FUNCTION_BLOCK FB_DataCollectionSequence
VAR
    iSystemCalibration : I_SystemCalibration;
    iResetSequence : I_ResetSequence;
    iTriggerManager : I_TriggerManager;

    eSequence : E_DataCollectionSequenceStep;
END_VAR


// Run our sequence here

CASE eSequence OF
    E_DataCollectionSequenceStep.WaitingForStart :
        // Do nothing

    E_DataCollectionSequenceStep.WaitingForInitialTrigger :

    E_DataCollectionSequenceStep.CalculateTimeToNextPoint :

    E_DataCollectionSequenceStep.AccelerateToScanningSpeed :

    E_DataCollectionSequenceStep.OperateAtScanningSpeedMakingMinuteAdjustments :

    E_DataCollectionSequenceStep.GoToNextRow :

    E_DataCollectionSequenceStep.WaitingForTriggerToStartNewRow :

    E_DataCollectionSequenceStep.Error :
        // Do nothing
    E_DataCollectionSequenceStep.Done :
        // Do nothing
END_CASE

//FB_Init is always available implicitly and it is used primarily for initialization.
//The return value is not evaluated. For a specific influence, you can also declare the
//methods explicitly and provide additional code there with the standard initialization
//code. You can evaluate the return value.
METHOD FB_Init: BOOL
VAR_INPUT
    bInitRetains: BOOL; // TRUE: the retain variables are initialized (reset warm / reset cold)
    bInCopyCode: BOOL;  // TRUE: the instance will be copied to the copy code afterward (online change)
    iSystemCalibration : I_SystemCalibration;
    iResetSequence : I_ResetSequence;
    iTriggerManager : I_TriggerManager;
END_VAR
THIS^.iSystemCalibration := iSystemCalibration;
THIS^.iResetSequence := iResetSequence;
THIS^.iTriggerManager := iTriggerManager;
END_METHOD

METHOD PRIVATE GetDataCollectionSequenceStep : E_DataCollectionSequenceStep
GetDataCollectionSequenceStep := THIS^.eSequence;
END_METHOD

METHOD PUBLIC IsRunningSequence : BOOL
IsRunningSequence := (GetDataCollectionSequenceStep() <> E_DataCollectionSequenceStep.WaitingForStart) AND
                     (GetDataCollectionSequenceStep() <> E_DataCollectionSequenceStep.Error) AND
                     (GetDataCollectionSequenceStep() <> E_DataCollectionSequenceStep.Done);
END_METHOD


METHOD PUBLIC Start
VAR_OUTPUT
    bError : BOOL;
    sErrorString : T_MaxString;
END_VAR

IF NOT iSystemCalibration.IsCalibrated() THEN
    bError := TRUE;
    sErrorString := 'Can$'t start data collection sequence. System is not calibrated';
    RETURN;
END_IF

IF NOT iResetSequence.IsReset() THEN
    bError := TRUE;
    sErrorString := 'Can$'t start data collection sequence. System is not reset';
    RETURN;
END_IF

IF eSequence <> E_DataCollectionSequenceStep.WaitingForStart AND eSequence <> E_DataCollectionSequenceStep.Error THEN
    bError := TRUE;
    sErrorString := 'Can$'t start data collection sequence. System is already running data collection sequence';
    RETURN;
END_IF

// Start the sequence
eSequence := E_DataCollectionSequenceStep.WaitingForInitialTrigger;
END_METHOD

END_FUNCTION_BLOCK

(* stored: Version 1.1.0.1
   POU FB_DataCollectionSequence: Id {ff4ff02d-226f-42e4-a962-43e0863e01e2}, SpecialFunc None
   Method FB_Init: Id {5079c59b-cf55-4794-bb0d-8c64eb0b5696}
   Method GetDataCollectionSequenceStep: Id {da174e3d-6bb1-47ea-84e1-708d7d51c1d7}
   Method IsRunningSequence: Id {ce51a9e7-106f-48b2-8628-a88f9b4221f0}
   Method Start: Id {f16f3bf4-22ce-4e24-96ce-7b48c13031de} *)
